(*********************************** G.D S.p.A. - Technical Department ***********************************
============= PROGRAM INFO ============
FOLDER:             TBD
MACHINES INVOLVED:  TBD 

============= DESCRIPTION =============
csp machine declaration

============= REVISIONS ===============
Date		Version	 	Author      	Description             
----------	-------		------------  	--------------------------------------------
2019/04/05 	0000.00	 	M.Grasso		Creation of the PRG

**********************************************************************************************************)
(*$R process_ref := prc; $*)
PROGRAM csp_case_tr_squaring_ls
VAR
	
	prc:											process;
	prc_path:										STRING;
	
END_VAR

_read_var_input();

_object_manager();

IF NOT objects_running()
THEN
	RETURN;	
END_IF

_read_process_image();

_mode_manager();

_set_runtime_properties();

(********************************* BODY *********************************)
(************************************************************************)

_handle_messages();

_write_output();

ACTION _handle_messages:
;
END_ACTION

ACTION _handle_process_test:
;
END_ACTION

ACTION _mode_manager:
IF process_mode_req_is_pending(prc)
THEN
    process_apply_mode_req_first_step(prc);
    CASE process_get_mode(prc) OF
        MODE_TO_ABSENT:
			;
        MODE_TO_INACTIVE:
			;
        MODE_TO_TEST:
			;
        MODE_TO_OPERATIONAL:
			;
    END_CASE
    process_apply_mode_req_second_step(prc);
END_IF
END_ACTION

ACTION _object_manager:
IF objects_initialization()
THEN
	sub_process_init(
		object_name					:= 'csp_case_tr_squaring_ls.prc', 
		process						:= csp_case_topRail_squaring.prc, 
		CONVERSION_this				:= prc);
		
	prc_path 						:= process_get_path(prc);
END_IF

IF objects_running()
THEN
	process_cycle(prc);
END_IF
END_ACTION

ACTION _read_process_image:
;
END_ACTION

ACTION _read_var_input:
;
END_ACTION

ACTION _set_runtime_properties:
;
END_ACTION

ACTION _write_output:
;
END_ACTION

END_PROGRAM

(* stored: Version 1.1.0.1, ProductVersion 3.1.4022.12
   POU csp_case_tr_squaring_ls: Id {6d730bab-db7e-4b39-997e-220dec2f3957}, SpecialFunc None
   Action _handle_messages: Id {69dc4ef1-e2c2-454f-a40b-4fc50dec75dc}
   Action _handle_process_test: Id {9d5409a2-5d43-4e6d-a741-51ddd31507b2}
   Action _mode_manager: Id {30a94e5f-f921-4e47-af40-e4d5cce1df7e}
   Action _object_manager: Id {749f0543-0b17-481c-96bd-ea43246cdcc4}
   Action _read_process_image: Id {7039c633-8452-41b8-986a-7159b0b5b127}
   Action _read_var_input: Id {0e9c056c-8d9f-4865-a7c4-cf0379902d15}
   Action _set_runtime_properties: Id {006b696c-daef-4f48-916b-a38e05dc3d5c}
   Action _write_output: Id {c9ceec1b-bb42-434e-a39c-a6dd3a2911bf} *)
